Universal Robots PolyScope program: 1234.urp

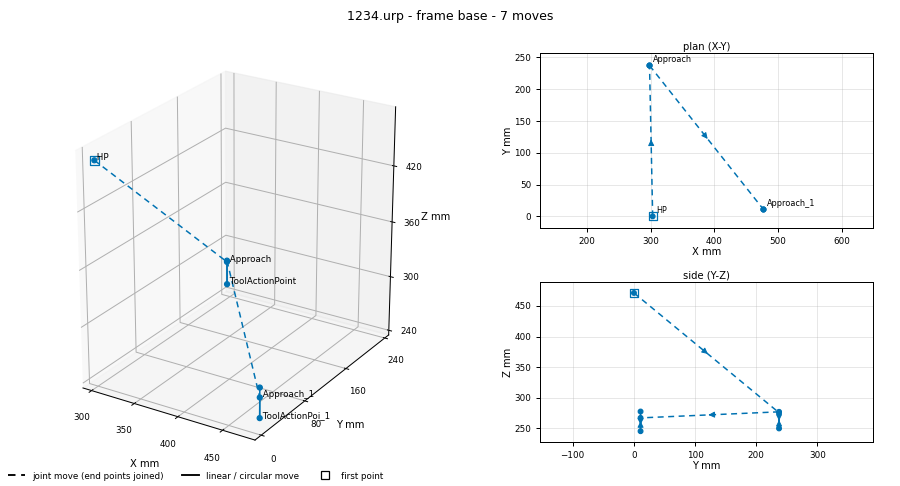
[picture p0: tool path of 1234.urp in frame base, 7 of 7 moves have a stored position in this frame; points joined in program order, loops and branches not executed]
Program 1234 (installation=default directory=/programs/Students createdIn=5.11.9.1010452 lastSavedIn=5.11.9.1010452 robotSerialNumber=20225200364)
Calibrated DH parameters: a=[0.00002, -0.569483, -0.54992, -0.00001, -0.000036, 0]; d=[0.180894, -146.691669, 192.918669, -46.053088, 0.119778, 0.115602]; alpha=[1.571425, -0.001534, 0.003359, 1.568739, -1.571477, 0]; deltaTheta=[0, 0.376258, -0.101074, -0.275185, -0.000002, 0]
Robot Program (runOnlyOnce=false)
  URCap RG Grip (OnRobot, OnRobot A/S) dataModel(rg-target-force=40.0, Variable(key=on_return, variable(name=on_return)))
  MoveJ speed 60 deg/s, acceleration 80 deg/s^2 (useActiveTCP=true) feature=Base
    Waypoint HP: TCP in base x=303.042 y=0.141 z=471.263 mm, rx=2.2261 ry=-2.2136 rz=-0.0016 rad; joints [35.103, -73.51, -125.081, -251.583, -90.244, -145.025] deg
    Loop Counting (count=3) loopVariable(name=Loop_1)
      URCap Palletizing (polyscope-pallet-impl, Universal Robots) dataModel(palletFeature=Base, isPalletizing=true, Variable(key=name, variable(name=Pallet_1)), Variable(key=globalCountingVariable, variable(name=Pallet_1_cnt_1, initializeExpression=1)), Variable(key=layerNumberVariable, variable(name=Pallet_1_lno, initializeExpression=1)), Variable(key=layerCountingVariable, variable(name=Pallet_1_lct, initializeExpression=1)), Variable(key=handleSeparatorVariable, variable(name=Pallet_1_sep, initializeExpression=False)), Variable(key=totalCountVariable, variable(name=Pallet_1_tct, initializeExpression=1)), Variable(key=referencePoint, variable(featureName=referencePoint)), Variable(key=separatorPoint, variable(featureName=separatorPoint)), Length(key=objectHeight value=0.00001 unit=M)); state(isChildrenLocked=true)
        URCap Patterns (polyscope-pallet-impl, Universal Robots) state(isChildrenLocked=true)
          URCap Pattern (polyscope-pallet-impl, Universal Robots) dataModel(UUID=e4365395-4c50-4ad8-b83e-2edba2ea2c24, patternType=LINE, objects=3, Variable(key=nameVariable, variable(name=Line_Pattern_1))); state(isChildrenLocked=true)
            URCap Item (polyscope-pallet-impl, Universal Robots) dataModel(UUID=0d25420d-b158-457f-940c-9220387c63c5, patternType=LINE, index=0, calibrationStatus=2, calibrationValidChecksum=true, calibrationDeltaTheta=[-2.1094217540068572E-7, 0.37625772532806073, -0.10107441100396769, -0.2751850025766889, -1.8024952768980196E-6, 2.9402326063437956E-8], calibrationA=[2.0416891277915125E-5, -0.5694828868469309, -0.5499202125525207, -9.504674691390763E-6, -3.603723657207661E-5, 0.0], calibrationD=[0.1808937726775539, -146.69166934821124, 192.91866861971778, -46.05308757405963, 0.11977780403821288, 0.11560212559305974], calibrationAlpha=[1.5714252480212174, -0.0015337665762078037, 0.0033588312559612306, 1.5687392298942362, -1.5714772428732047, 0.0], calibrationJointChecksum=[-1490546360, -1456574554, -1506622700, -1493399207, -1492840923, -1492940558], baseToFeature=[0.0, 0.0, 0.0, 0.0, 0.0, 0.0], TCPOffset=[1.0322624480613163E-5, -1.0290119388300933E-5, -7.776170349860223E-7, -1.6607002647202897E-5, -3.763130106398986E-5, 4.268658811272661E-5], Variable(key=variable, variable(name=StartItem_1)), JointPositions(key=jointpositions, JointPosition(key=[1], Angle(key=pos value=1.147015 unit=RAD)), JointPosition(key=[2], Angle(key=pos value=-1.693616 unit=RAD)), JointPosition(key=[3], Angle(key=pos value=-2.283738 unit=RAD)), JointPosition(key=[4], Angle(key=pos value=-3.879032 unit=RAD)), JointPosition(key=[5], Angle(key=pos value=-1.575117 unit=RAD)), JointPosition(key=[6], Angle(key=pos value=-1.994873 unit=RAD))))
            URCap Item (polyscope-pallet-impl, Universal Robots) dataModel(UUID=9305f81a-3f95-4564-bffa-4e46a6b45f4b, patternType=LINE, index=1, calibrationStatus=2, calibrationValidChecksum=true, calibrationDeltaTheta=[-2.1094217540068572E-7, 0.37625772532806073, -0.10107441100396769, -0.2751850025766889, -1.8024952768980196E-6, 2.9402326063437956E-8], calibrationA=[2.0416891277915125E-5, -0.5694828868469309, -0.5499202125525207, -9.504674691390763E-6, -3.603723657207661E-5, 0.0], calibrationD=[0.1808937726775539, -146.69166934821124, 192.91866861971778, -46.05308757405963, 0.11977780403821288, 0.11560212559305974], calibrationAlpha=[1.5714252480212174, -0.0015337665762078037, 0.0033588312559612306, 1.5687392298942362, -1.5714772428732047, 0.0], calibrationJointChecksum=[-1490546360, -1456574554, -1506622700, -1493399207, -1492840923, -1492940558], baseToFeature=[0.0, 0.0, 0.0, 0.0, 0.0, 0.0], TCPOffset=[-1.3170302495285613E-5, -1.9800938602099194E-5, -1.0039190083632743E-5, 3.3348788237127763E-5, 3.2467099588180865E-6, 4.129712166360907E-5], Variable(key=variable, variable(name=EndItem_1)), JointPositions(key=jointpositions, JointPosition(key=[1], Angle(key=pos value=1.297552 unit=RAD)), JointPosition(key=[2], Angle(key=pos value=-1.625682 unit=RAD)), JointPosition(key=[3], Angle(key=pos value=-2.356941 unit=RAD)), JointPosition(key=[4], Angle(key=pos value=-3.873484 unit=RAD)), JointPosition(key=[5], Angle(key=pos value=-1.575448 unit=RAD)), JointPosition(key=[6], Angle(key=pos value=-1.84435 unit=RAD))))
        URCap Layers (polyscope-pallet-impl, Universal Robots) dataModel(separators=[false], selectedPatterns=[e4365395-4c50-4ad8-b83e-2edba2ea2c24])
        URCap At Each Item (polyscope-pallet-impl, Universal Robots) dataModel(selectedPattern=e4365395-4c50-4ad8-b83e-2edba2ea2c24, selectedPosition=0d25420d-b158-457f-940c-9220387c63c5, Approach_calibrationDeltaTheta=[-2.1094217540068572E-7, 0.37625772532806073, -0.10107441100396769, -0.2751850025766889, -1.8024952768980196E-6, 2.9402326063437956E-8], Approach_calibrationA=[2.0416891277915125E-5, -0.5694828868469309, -0.5499202125525207, -9.504674691390763E-6, -3.603723657207661E-5, 0.0], Approach_calibrationD=[0.1808937726775539, -146.69166934821124, 192.91866861971778, -46.05308757405963, 0.11977780403821288, 0.11560212559305974], Approach_calibrationAlpha=[1.5714252480212174, -0.0015337665762078037, 0.0033588312559612306, 1.5687392298942362, -1.5714772428732047, 0.0], Approach_calibrationJointChecksum=[-1490546360, -1456574554, -1506622700, -1493399207, -1492840923, -1492940558], Approach_calibrationStatus=2, Approach_calibrationValidChecksum=true, Approach_baseToFeature=[0.0, 0.0, 0.0, 0.0, 0.0, 0.0], Approach_TCPOffset=[1.4910819420399513E-5, 1.4596702744229528E-5, 7.489766990720348E-6, 9.713365963077813E-6, 2.2921076932334492E-5, -3.1189236069694936E-5], Exit_calibrationDeltaTheta=[-2.1094217540068572E-7, 0.37625772532806073, -0.10107441100396769, -0.2751850025766889, -1.8024952768980196E-6, 2.9402326063437956E-8], Exit_calibrationA=[2.0416891277915125E-5, -0.5694828868469309, -0.5499202125525207, -9.504674691390763E-6, -3.603723657207661E-5, 0.0], Exit_calibrationD=[0.1808937726775539, -146.69166934821124, 192.91866861971778, -46.05308757405963, 0.11977780403821288, 0.11560212559305974], Exit_calibrationAlpha=[1.5714252480212174, -0.0015337665762078037, 0.0033588312559612306, 1.5687392298942362, -1.5714772428732047, 0.0], Exit_calibrationJointChecksum=[-1490546360, -1456574554, -1506622700, -1493399207, -1492840923, -1492940558], Exit_calibrationStatus=2, Exit_calibrationValidChecksum=true, Exit_baseToFeature=[0.0, 0.0, 0.0, 0.0, 0.0, 0.0], Exit_TCPOffset=[6.060465969015549E-6, 9.910566535209497E-7, 2.489721756221419E-5, -6.630066338378124E-6, 7.042242020715943E-5, -7.850838662992361E-6], currentWizardState=SHOW_DONE, Pose(key=refBaseToFeature, Position(key=posePosition, Length(key=X value=0 unit=M), Length(key=Y value=0 unit=M), Length(key=Z value=0 unit=M)), Rotation(key=poseRotation, Angle(key=RX value=0 unit=RAD), Angle(key=RY value=0 unit=RAD), Angle(key=RZ value=0 unit=RAD))), Pose(key=refPose, Position(key=posePosition, Length(key=X value=0.298115 unit=M), Length(key=Y value=0.23722 unit=M), Length(key=Z value=0.249864 unit=M)), Rotation(key=poseRotation, Angle(key=RX value=2.226048 unit=RAD), Angle(key=RY value=-2.21368 unit=RAD), Angle(key=RZ value=-0.001626 unit=RAD))), JointPositions(key=Approach_jointpositions, JointPosition(key=[1], Angle(key=pos value=1.146903 unit=RAD)), JointPosition(key=[2], Angle(key=pos value=-1.653942 unit=RAD)), JointPosition(key=[3], Angle(key=pos value=-2.264714 unit=RAD)), JointPosition(key=[4], Angle(key=pos value=-3.937702 unit=RAD)), JointPosition(key=[5], Angle(key=pos value=-1.575306 unit=RAD)), JointPosition(key=[6], Angle(key=pos value=-1.995129 unit=RAD))), JointPositions(key=Exit_jointpositions, JointPosition(key=[1], Angle(key=pos value=1.146899 unit=RAD)), JointPosition(key=[2], Angle(key=pos value=-1.651818 unit=RAD)), JointPosition(key=[3], Angle(key=pos value=-2.263592 unit=RAD)), JointPosition(key=[4], Angle(key=pos value=-3.940949 unit=RAD)), JointPosition(key=[5], Angle(key=pos value=-1.575314 unit=RAD)), JointPosition(key=[6], Angle(key=pos value=-1.995143 unit=RAD))))
          URCap Generated Movements (polyscope-pallet-impl, Universal Robots) state(isChildrenLocked=true)
            MoveJ speed 60 deg/s, acceleration 80 deg/s^2 (useActiveTCP=true) feature=referencePoint
              Waypoint Approach: TCP in base x=298.1 y=237.205 z=275.587 mm, rx=2.2261 ry=-2.2136 rz=-0.0016 rad; joints [65.714, -94.763, -129.761, -225.613, -90.257, -114.313] deg; TCP offset x=0 y=0 z=0 mm, rx=0 ry=0 rz=0 rad; feature pose in base x=298.105 y=237.231 z=267.615 mm, rx=2.2261 ry=-2.2136 rz=-0.0016 rad
            MoveL speed 250 mm/s, acceleration 1200 mm/s^2 (useActiveTCP=true) feature(featureName=referencePoint)
              Waypoint ToolActionPoint: TCP in base x=298.115 y=237.22 z=249.864 mm, rx=2.226 ry=-2.2137 rz=-0.0016 rad; joints [65.716, -97.037, -130.848, -222.251, -90.249, -114.298] deg; TCP offset x=0 y=0 z=0 mm, rx=0 ry=0 rz=0 rad
            Folder Tool action
              URCap RG Grip (OnRobot, OnRobot A/S) dataModel(rg-target-force=40.0, rg-target-width=0.075)
            MoveL speed 250 mm/s, acceleration 1200 mm/s^2 (useActiveTCP=true) feature(featureName=referencePoint)
              Waypoint Exit_1: TCP in base x=298.114 y=237.214 z=277.003 mm, rx=2.226 ry=-2.2136 rz=-0.0016 rad; joints [65.713, -94.645, -129.696, -225.799, -90.258, -114.314] deg; TCP offset x=0 y=0 z=0 mm, rx=0 ry=0 rz=0 rad
      URCap Palletizing (polyscope-pallet-impl, Universal Robots) dataModel(palletFeature=Base, isPalletizing=true, Variable(key=name, variable(name=Pallet_2)), Variable(key=globalCountingVariable, variable(name=Pallet_2_cnt, initializeExpression=1)), Variable(key=layerNumberVariable, variable(name=Pallet_2_lno, initializeExpression=1)), Variable(key=layerCountingVariable, variable(name=Pallet_2_lct, initializeExpression=1)), Variable(key=handleSeparatorVariable, variable(name=Pallet_2_sep, initializeExpression=False)), Variable(key=totalCountVariable, variable(name=Pallet_2_tct, initializeExpression=1)), Variable(key=referencePoint, variable(featureName=referencePoin_1)), Variable(key=separatorPoint, variable(featureName=separatorPoin_1)), Length(key=objectHeight value=0.00001 unit=M)); state(isChildrenLocked=true)
        URCap Patterns (polyscope-pallet-impl, Universal Robots) state(isChildrenLocked=true)
          URCap Pattern (polyscope-pallet-impl, Universal Robots) dataModel(UUID=385f3494-e727-448f-a127-f77b145563ee, patternType=LINE, objects=3, Variable(key=nameVariable, variable(name=Line_Pattern_2))); state(isChildrenLocked=true)
            URCap Item (polyscope-pallet-impl, Universal Robots) dataModel(UUID=34ea186d-f35e-4bf0-bbd3-d250248905ab, patternType=LINE, index=0, calibrationDeltaTheta=[-2.1094217540068572E-7, 0.37625772532806073, -0.10107441100396769, -0.2751850025766889, -1.8024952768980196E-6, 2.9402326063437956E-8], calibrationA=[2.0416891277915125E-5, -0.5694828868469309, -0.5499202125525207, -9.504674691390763E-6, -3.603723657207661E-5, 0.0], calibrationD=[0.1808937726775539, -146.69166934821124, 192.91866861971778, -46.05308757405963, 0.11977780403821288, 0.11560212559305974], calibrationAlpha=[1.5714252480212174, -0.0015337665762078037, 0.0033588312559612306, 1.5687392298942362, -1.5714772428732047, 0.0], calibrationJointChecksum=[-1490546360, -1456574554, -1506622700, -1493399207, -1492840923, -1492940558], calibrationStatus=2, calibrationValidChecksum=true, baseToFeature=[0.0, 0.0, 0.0, 0.0, 0.0, 0.0], TCPOffset=[-1.2379940612921615E-5, -5.411534380939109E-6, 1.4314669030096594E-5, 1.2869323820080988E-5, -2.7560022474741347E-5, -2.026789760782582E-5], Variable(key=variable, variable(name=StartItem_2)), JointPositions(key=jointpositions, JointPosition(key=[1], Angle(key=pos value=0.396635 unit=RAD)), JointPosition(key=[2], Angle(key=pos value=-1.845251 unit=RAD)), JointPosition(key=[3], Angle(key=pos value=-2.096918 unit=RAD)), JointPosition(key=[4], Angle(key=pos value=-3.914957 unit=RAD)), JointPosition(key=[5], Angle(key=pos value=-1.572949 unit=RAD)), JointPosition(key=[6], Angle(key=pos value=-2.75418 unit=RAD))))
            URCap Item (polyscope-pallet-impl, Universal Robots) dataModel(UUID=ed631416-e6be-4585-b411-f4ccb5116b81, patternType=LINE, index=1, calibrationDeltaTheta=[-2.1094217540068572E-7, 0.37625772532806073, -0.10107441100396769, -0.2751850025766889, -1.8024952768980196E-6, 2.9402326063437956E-8], calibrationA=[2.0416891277915125E-5, -0.5694828868469309, -0.5499202125525207, -9.504674691390763E-6, -3.603723657207661E-5, 0.0], calibrationD=[0.1808937726775539, -146.69166934821124, 192.91866861971778, -46.05308757405963, 0.11977780403821288, 0.11560212559305974], calibrationAlpha=[1.5714252480212174, -0.0015337665762078037, 0.0033588312559612306, 1.5687392298942362, -1.5714772428732047, 0.0], calibrationJointChecksum=[-1490546360, -1456574554, -1506622700, -1493399207, -1492840923, -1492940558], calibrationStatus=2, calibrationValidChecksum=true, baseToFeature=[0.0, 0.0, 0.0, 0.0, 0.0, 0.0], TCPOffset=[1.5692351169462743E-5, 2.7434884057320197E-5, 2.1610494246870893E-7, 7.47530793387282E-6, -2.5011070988082327E-5, 1.9719414038610633E-5], Variable(key=variable, variable(name=EndItem_2)), JointPositions(key=jointpositions, JointPosition(key=[1], Angle(key=pos value=0.444688 unit=RAD)), JointPosition(key=[2], Angle(key=pos value=-1.774252 unit=RAD)), JointPosition(key=[3], Angle(key=pos value=-2.194163 unit=RAD)), JointPosition(key=[4], Angle(key=pos value=-3.888722 unit=RAD)), JointPosition(key=[5], Angle(key=pos value=-1.57313 unit=RAD)), JointPosition(key=[6], Angle(key=pos value=-2.706067 unit=RAD))))
        URCap Layers (polyscope-pallet-impl, Universal Robots) dataModel(separators=[false], selectedPatterns=[385f3494-e727-448f-a127-f77b145563ee])
        URCap At Each Item (polyscope-pallet-impl, Universal Robots) dataModel(selectedPattern=385f3494-e727-448f-a127-f77b145563ee, selectedPosition=34ea186d-f35e-4bf0-bbd3-d250248905ab, Approach_calibrationDeltaTheta=[-2.1094217540068572E-7, 0.37625772532806073, -0.10107441100396769, -0.2751850025766889, -1.8024952768980196E-6, 2.9402326063437956E-8], Approach_calibrationA=[2.0416891277915125E-5, -0.5694828868469309, -0.5499202125525207, -9.504674691390763E-6, -3.603723657207661E-5, 0.0], Approach_calibrationD=[0.1808937726775539, -146.69166934821124, 192.91866861971778, -46.05308757405963, 0.11977780403821288, 0.11560212559305974], Approach_calibrationAlpha=[1.5714252480212174, -0.0015337665762078037, 0.0033588312559612306, 1.5687392298942362, -1.5714772428732047, 0.0], Approach_calibrationJointChecksum=[-1490546360, -1456574554, -1506622700, -1493399207, -1492840923, -1492940558], Approach_calibrationStatus=2, Approach_calibrationValidChecksum=true, Approach_baseToFeature=[0.0, 0.0, 0.0, 0.0, 0.0, 0.0], Approach_TCPOffset=[-1.1558175415270471E-5, -2.1860093043946094E-5, 1.4099419648916367E-5, 3.835355430658518E-5, -9.325815871687334E-6, -3.319324898755077E-5], Exit_calibrationDeltaTheta=[-2.1094217540068572E-7, 0.37625772532806073, -0.10107441100396769, -0.2751850025766889, -1.8024952768980196E-6, 2.9402326063437956E-8], Exit_calibrationA=[2.0416891277915125E-5, -0.5694828868469309, -0.5499202125525207, -9.504674691390763E-6, -3.603723657207661E-5, 0.0], Exit_calibrationD=[0.1808937726775539, -146.69166934821124, 192.91866861971778, -46.05308757405963, 0.11977780403821288, 0.11560212559305974], Exit_calibrationAlpha=[1.5714252480212174, -0.0015337665762078037, 0.0033588312559612306, 1.5687392298942362, -1.5714772428732047, 0.0], Exit_calibrationJointChecksum=[-1490546360, -1456574554, -1506622700, -1493399207, -1492840923, -1492940558], Exit_calibrationStatus=2, Exit_calibrationValidChecksum=true, Exit_baseToFeature=[0.0, 0.0, 0.0, 0.0, 0.0, 0.0], Exit_TCPOffset=[-6.555920474158802E-6, -1.5192608014691356E-5, 8.35285353906201E-6, 5.871992185230492E-6, -7.41037084393287E-5, -2.072878691388236E-7], currentWizardState=LANDING, Pose(key=refBaseToFeature, Position(key=posePosition, Length(key=X value=0 unit=M), Length(key=Y value=0 unit=M), Length(key=Z value=0 unit=M)), Rotation(key=poseRotation, Angle(key=RX value=0 unit=RAD), Angle(key=RY value=0 unit=RAD), Angle(key=RZ value=0 unit=RAD))), Pose(key=refPose, Position(key=posePosition, Length(key=X value=0.477175 unit=M), Length(key=Y value=0.010932 unit=M), Length(key=Z value=0.245346 unit=M)), Rotation(key=poseRotation, Angle(key=RX value=2.23581 unit=RAD), Angle(key=RY value=-2.203617 unit=RAD), Angle(key=RZ value=-0.001099 unit=RAD))), JointPositions(key=Approach_jointpositions, JointPosition(key=[1], Angle(key=pos value=0.396626 unit=RAD)), JointPosition(key=[2], Angle(key=pos value=-1.816549 unit=RAD)), JointPosition(key=[3], Angle(key=pos value=-2.083253 unit=RAD)), JointPosition(key=[4], Angle(key=pos value=-3.957302 unit=RAD)), JointPosition(key=[5], Angle(key=pos value=-1.573081 unit=RAD)), JointPosition(key=[6], Angle(key=pos value=-2.75434 unit=RAD))), JointPositions(key=Exit_jointpositions, JointPosition(key=[1], Angle(key=pos value=0.396613 unit=RAD)), JointPosition(key=[2], Angle(key=pos value=-1.803352 unit=RAD)), JointPosition(key=[3], Angle(key=pos value=-2.076219 unit=RAD)), JointPosition(key=[4], Angle(key=pos value=-3.977533 unit=RAD)), JointPosition(key=[5], Angle(key=pos value=-1.573132 unit=RAD)), JointPosition(key=[6], Angle(key=pos value=-2.754416 unit=RAD))))
          URCap Generated Movements (polyscope-pallet-impl, Universal Robots) state(isChildrenLocked=true)
            MoveJ speed 60 deg/s, acceleration 80 deg/s^2 (useActiveTCP=true) feature=referencePoin_1
              Waypoint Approach_1: TCP in base x=477.197 y=10.944 z=267.103 mm, rx=2.2359 ry=-2.2036 rz=-0.0011 rad; joints [22.725, -104.083, -119.36, -226.734, -90.131, -157.814] deg; TCP offset x=0 y=0 z=0 mm, rx=0 ry=0 rz=0 rad; feature pose in base x=477.175 y=10.932 z=245.346 mm, rx=2.2358 ry=-2.2036 rz=-0.0011 rad
            MoveL speed 250 mm/s, acceleration 1200 mm/s^2 (useActiveTCP=true) feature(featureName=referencePoin_1)
              Waypoint ToolActionPoi_1: TCP in base x=477.175 y=10.932 z=245.346 mm, rx=2.2358 ry=-2.2036 rz=-0.0011 rad; joints [22.726, -105.726, -120.145, -224.308, -90.125, -157.803] deg; TCP offset x=0 y=0 z=0 mm, rx=0 ry=0 rz=0 rad
            Folder Tool action
              URCap RG Grip (OnRobot, OnRobot A/S) dataModel(rg-target-force=40.0)
            MoveL speed 250 mm/s, acceleration 1200 mm/s^2 (useActiveTCP=true) feature(featureName=referencePoin_1)
              Waypoint Exit_2: TCP in base x=477.19 y=10.939 z=277.506 mm, rx=2.2359 ry=-2.2037 rz=-0.0012 rad; joints [22.723, -103.326, -118.957, -227.894, -90.138, -157.817] deg; TCP offset x=0 y=0 z=0 mm, rx=0 ry=0 rz=0 rad
